// TIA Portal V21 export
TYPE "Tra_Formato"
   STRUCT
      Nome_1 { S7_SetPoint := 'True'} : String[30];
      "Diam.Cont.Riemp.1" { S7_SetPoint := 'True'} : Real;   // Diametro contenitore riempitrice 1 [mm]
      "Diam.Cont.Riemp.2" { S7_SetPoint := 'True'} : Real;   // Diametro contenitore riempitrice 1 [mm]
   END_STRUCT;
END_TYPE
